//Enumeration for Machineunits
TYPE E_UnitName :
(
	eMachine		:= 1,
	eSeperation		:= 2,
	eEjectorPlastic	:= 3,
	eAxisMain		:= 4,
	eEjectorMetal	:= 5,
	eSensorPlastic	:= 6,
	eAxisPlastic	:= 7,
	eSensorMetal	:= 8,
	eAxisMetal		:= 9
)DINT;
END_TYPE

(* stored: Version 1.1.0.1, ProductVersion 3.1.4018.5
   DUT E_UnitName: Id {38fb3a11-736e-4cc8-89e9-4c4bd7e49aca} *)
